// MAIN was replaced by EventTracker and DelayTracker
PROGRAM MAIN_DEPRECATED
VAR
    placeholder : BOOL := FALSE;
END_VAR

// This POU is deprecated. Use EventTracker and DelayTracker instead.
placeholder := placeholder;

END_PROGRAM

(* stored: Version 1.1.0.1, ProductVersion 3.1.4024.15
   POU MAIN: Id {074e3488-9984-4e9d-a106-00737da1eebc}, SpecialFunc None *)
